// TIA Portal V19 export
FUNCTION "MODE" : Void   // FC3, LAD
{ S7_Optimized_Access := 'TRUE' }
// stored: SetENOAutomatically false
   VAR_TEMP   // added for the SCL form of the ladder/FBD networks
      _w1 : Bool;
   END_VAR
BEGIN

REGION Network 1: MANUAL_MODE_SELECTION
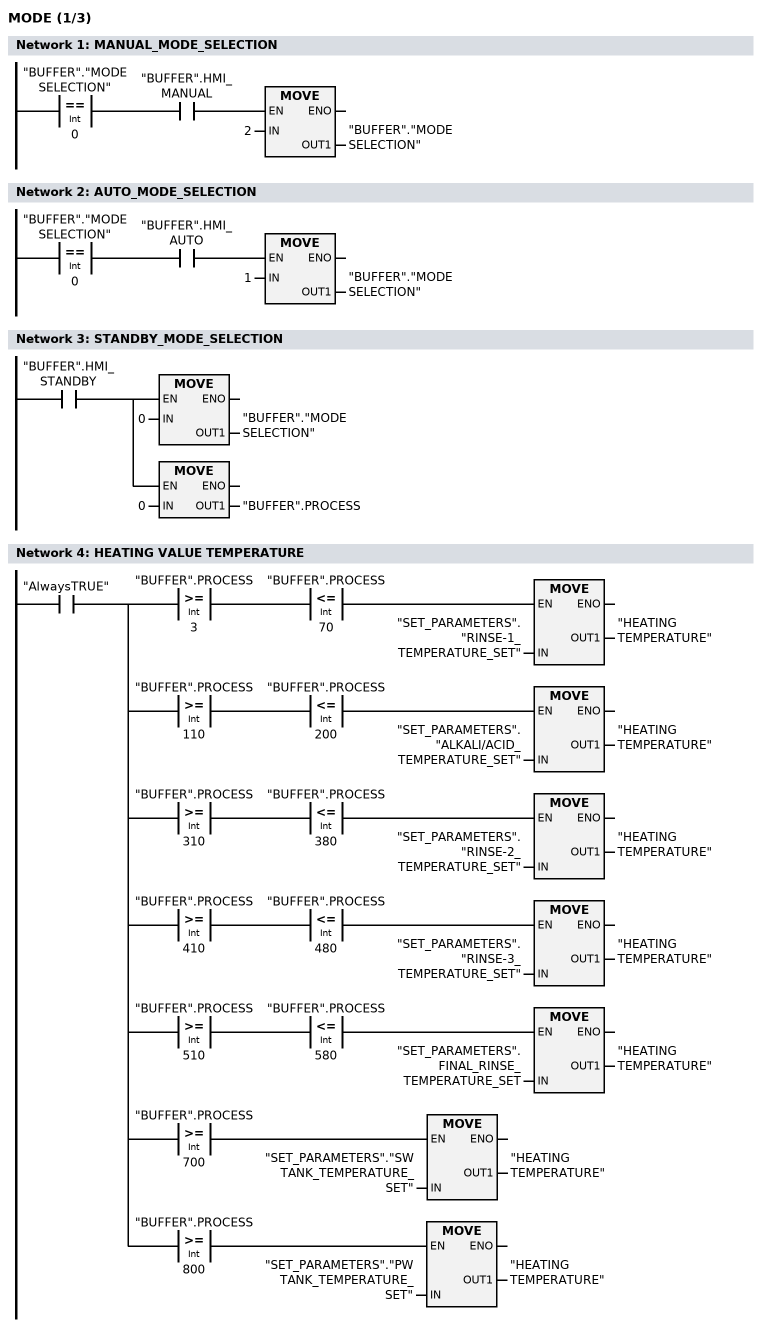
   RUNG wire#powerrail
      { S7_Templates := "SrcType := Int" } EQ_Contact(in1 := "BUFFER"."MODE SELECTION", in2 := 0)
      Contact( "BUFFER".HMI_MANUAL )
      Move(in := 2, out1 => "BUFFER"."MODE SELECTION")
   END_RUNG
   // the same network as SCL:
   IF ("BUFFER"."MODE SELECTION" = 0) AND "BUFFER".HMI_MANUAL THEN "BUFFER"."MODE SELECTION" := 2; END_IF;
END_REGION

REGION Network 2: AUTO_MODE_SELECTION
   RUNG wire#powerrail
      { S7_Templates := "SrcType := Int" } EQ_Contact(in1 := "BUFFER"."MODE SELECTION", in2 := 0)
      Contact( "BUFFER".HMI_AUTO )
      Move(in := 1, out1 => "BUFFER"."MODE SELECTION")
   END_RUNG
   // the same network as SCL:
   IF ("BUFFER"."MODE SELECTION" = 0) AND "BUFFER".HMI_AUTO THEN "BUFFER"."MODE SELECTION" := 1; END_IF;
END_REGION

REGION Network 3: STANDBY_MODE_SELECTION
   RUNG wire#powerrail
      Contact( "BUFFER".HMI_STANDBY )
      wire#w1
      Move(in := 0, out1 => "BUFFER"."MODE SELECTION")
   END_RUNG
   RUNG wire#w1
      Move(in := 0, out1 => "BUFFER".PROCESS)
   END_RUNG
   // the same network as SCL:
   IF "BUFFER".HMI_STANDBY THEN
       "BUFFER"."MODE SELECTION" := 0;
       "BUFFER".PROCESS := 0;
   END_IF;
END_REGION

REGION Network 4: HEATING VALUE TEMPERATURE
   RUNG wire#powerrail
      Contact( "AlwaysTRUE" )
      wire#w1
      { S7_Templates := "SrcType := Int" } GE_Contact(in1 := "BUFFER".PROCESS, in2 := 3)
      { S7_Templates := "SrcType := Int" } LE_Contact(in1 := "BUFFER".PROCESS, in2 := 70)
      Move(in := "SET_PARAMETERS"."RINSE-1_TEMPERATURE_SET", out1 => "HEATING TEMPERATURE")
   END_RUNG
   RUNG wire#w1
      { S7_Templates := "SrcType := Int" } GE_Contact(in1 := "BUFFER".PROCESS, in2 := 110)
      { S7_Templates := "SrcType := Int" } LE_Contact(in1 := "BUFFER".PROCESS, in2 := 200)
      Move(in := "SET_PARAMETERS"."ALKALI/ACID_TEMPERATURE_SET", out1 => "HEATING TEMPERATURE")
   END_RUNG
   RUNG wire#w1
      { S7_Templates := "SrcType := Int" } GE_Contact(in1 := "BUFFER".PROCESS, in2 := 310)
      { S7_Templates := "SrcType := Int" } LE_Contact(in1 := "BUFFER".PROCESS, in2 := 380)
      Move(in := "SET_PARAMETERS"."RINSE-2_TEMPERATURE_SET", out1 => "HEATING TEMPERATURE")
   END_RUNG
   RUNG wire#w1
      { S7_Templates := "SrcType := Int" } GE_Contact(in1 := "BUFFER".PROCESS, in2 := 410)
      { S7_Templates := "SrcType := Int" } LE_Contact(in1 := "BUFFER".PROCESS, in2 := 480)
      Move(in := "SET_PARAMETERS"."RINSE-3_TEMPERATURE_SET", out1 => "HEATING TEMPERATURE")
   END_RUNG
   RUNG wire#w1
      { S7_Templates := "SrcType := Int" } GE_Contact(in1 := "BUFFER".PROCESS, in2 := 510)
      { S7_Templates := "SrcType := Int" } LE_Contact(in1 := "BUFFER".PROCESS, in2 := 580)
      Move(in := "SET_PARAMETERS".FINAL_RINSE_TEMPERATURE_SET, out1 => "HEATING TEMPERATURE")
   END_RUNG
   RUNG wire#w1
      { S7_Templates := "SrcType := Int" } GE_Contact(in1 := "BUFFER".PROCESS, in2 := 700)
      Move(in := "SET_PARAMETERS"."SW TANK_TEMPERATURE_SET", out1 => "HEATING TEMPERATURE")
   END_RUNG
   RUNG wire#w1
      { S7_Templates := "SrcType := Int" } GE_Contact(in1 := "BUFFER".PROCESS, in2 := 800)
      Move(in := "SET_PARAMETERS"."PW TANK_TEMPERATURE_SET", out1 => "HEATING TEMPERATURE")
   END_RUNG
   // the same network as SCL:
   IF "AlwaysTRUE" AND ("BUFFER".PROCESS >= 3) AND ("BUFFER".PROCESS <= 70) THEN
       "HEATING TEMPERATURE" := "SET_PARAMETERS"."RINSE-1_TEMPERATURE_SET";
   END_IF;
   IF "AlwaysTRUE" AND ("BUFFER".PROCESS >= 110) AND ("BUFFER".PROCESS <= 200) THEN
       "HEATING TEMPERATURE" := "SET_PARAMETERS"."ALKALI/ACID_TEMPERATURE_SET";
   END_IF;
   IF "AlwaysTRUE" AND ("BUFFER".PROCESS >= 310) AND ("BUFFER".PROCESS <= 380) THEN
       "HEATING TEMPERATURE" := "SET_PARAMETERS"."RINSE-2_TEMPERATURE_SET";
   END_IF;
   IF "AlwaysTRUE" AND ("BUFFER".PROCESS >= 410) AND ("BUFFER".PROCESS <= 480) THEN
       "HEATING TEMPERATURE" := "SET_PARAMETERS"."RINSE-3_TEMPERATURE_SET";
   END_IF;
   IF "AlwaysTRUE" AND ("BUFFER".PROCESS >= 510) AND ("BUFFER".PROCESS <= 580) THEN
       "HEATING TEMPERATURE" := "SET_PARAMETERS".FINAL_RINSE_TEMPERATURE_SET;
   END_IF;
   IF "AlwaysTRUE" AND ("BUFFER".PROCESS >= 700) THEN
       "HEATING TEMPERATURE" := "SET_PARAMETERS"."SW TANK_TEMPERATURE_SET";
   END_IF;
   IF "AlwaysTRUE" AND ("BUFFER".PROCESS >= 800) THEN
       "HEATING TEMPERATURE" := "SET_PARAMETERS"."PW TANK_TEMPERATURE_SET";
   END_IF;
END_REGION

REGION Network 5: HEATING HYSTERSIS
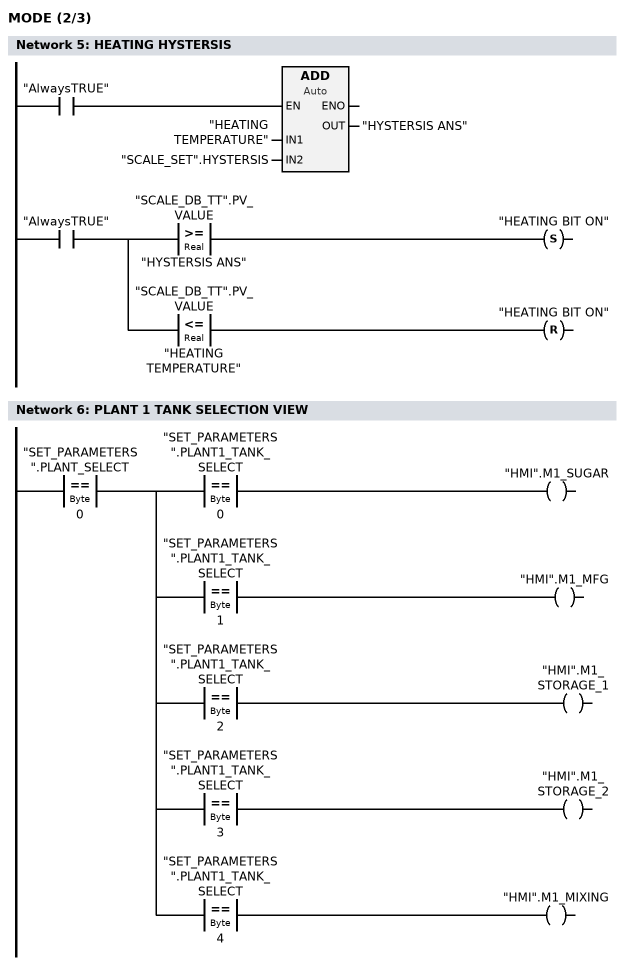
   RUNG wire#powerrail
      Contact( "AlwaysTRUE" )
      Add(in1 := "HEATING TEMPERATURE", in2 := "SCALE_SET".HYSTERSIS, out => "HYSTERSIS ANS")
   END_RUNG
   RUNG wire#powerrail
      Contact( "AlwaysTRUE" )
      wire#w1
      { S7_Templates := "SrcType := Real" } GE_Contact(in1 := "SCALE_DB_TT".PV_VALUE, in2 := "HYSTERSIS ANS")
      S_Coil( "HEATING BIT ON" )
   END_RUNG
   RUNG wire#w1
      { S7_Templates := "SrcType := Real" } LE_Contact(in1 := "SCALE_DB_TT".PV_VALUE, in2 := "HEATING TEMPERATURE")
      R_Coil( "HEATING BIT ON" )
   END_RUNG
   // the same network as SCL:
   IF "AlwaysTRUE" THEN "HYSTERSIS ANS" := "HEATING TEMPERATURE" + "SCALE_SET".HYSTERSIS; END_IF;
   IF "AlwaysTRUE" AND ("SCALE_DB_TT".PV_VALUE >= "HYSTERSIS ANS") THEN "HEATING BIT ON" := TRUE; END_IF;
   IF "AlwaysTRUE" AND ("SCALE_DB_TT".PV_VALUE <= "HEATING TEMPERATURE") THEN
       "HEATING BIT ON" := FALSE;
   END_IF;
END_REGION

REGION Network 6: PLANT 1 TANK SELECTION VIEW
   RUNG wire#powerrail
      { S7_Templates := "SrcType := Byte" } EQ_Contact(in1 := "SET_PARAMETERS".PLANT_SELECT, in2 := 0)
      wire#w1
      { S7_Templates := "SrcType := Byte" } EQ_Contact(in1 := "SET_PARAMETERS".PLANT1_TANK_SELECT, in2 := 0)
      Coil( "HMI".M1_SUGAR )
   END_RUNG
   RUNG wire#w1
      { S7_Templates := "SrcType := Byte" } EQ_Contact(in1 := "SET_PARAMETERS".PLANT1_TANK_SELECT, in2 := 1)
      Coil( "HMI".M1_MFG )
   END_RUNG
   RUNG wire#w1
      { S7_Templates := "SrcType := Byte" } EQ_Contact(in1 := "SET_PARAMETERS".PLANT1_TANK_SELECT, in2 := 2)
      Coil( "HMI".M1_STORAGE_1 )
   END_RUNG
   RUNG wire#w1
      { S7_Templates := "SrcType := Byte" } EQ_Contact(in1 := "SET_PARAMETERS".PLANT1_TANK_SELECT, in2 := 3)
      Coil( "HMI".M1_STORAGE_2 )
   END_RUNG
   RUNG wire#w1
      { S7_Templates := "SrcType := Byte" } EQ_Contact(in1 := "SET_PARAMETERS".PLANT1_TANK_SELECT, in2 := 4)
      Coil( "HMI".M1_MIXING )
   END_RUNG
   // the same network as SCL:
   #_w1 := "SET_PARAMETERS".PLANT_SELECT = 0;
   "HMI".M1_SUGAR := #_w1 AND ("SET_PARAMETERS".PLANT1_TANK_SELECT = 0);
   "HMI".M1_MFG := #_w1 AND ("SET_PARAMETERS".PLANT1_TANK_SELECT = 1);
   "HMI".M1_STORAGE_1 := #_w1 AND ("SET_PARAMETERS".PLANT1_TANK_SELECT = 2);
   "HMI".M1_STORAGE_2 := #_w1 AND ("SET_PARAMETERS".PLANT1_TANK_SELECT = 3);
   "HMI".M1_MIXING := #_w1 AND ("SET_PARAMETERS".PLANT1_TANK_SELECT = 4);
END_REGION

REGION Network 7: PLANT 2 TANK SELECTION VIEW
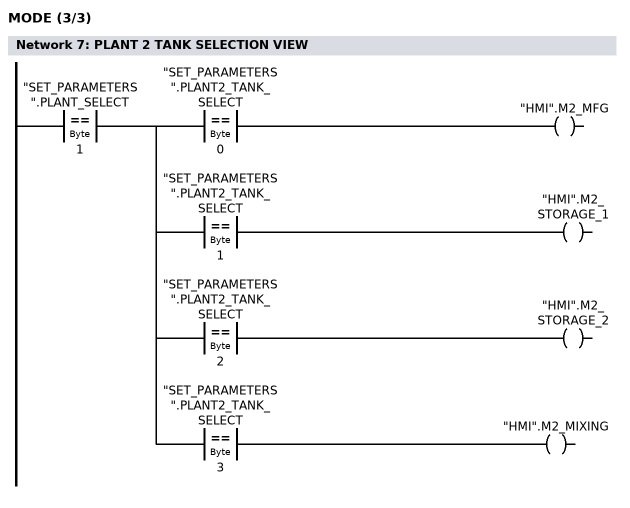
   RUNG wire#powerrail
      { S7_Templates := "SrcType := Byte" } EQ_Contact(in1 := "SET_PARAMETERS".PLANT_SELECT, in2 := 1)
      wire#w1
      { S7_Templates := "SrcType := Byte" } EQ_Contact(in1 := "SET_PARAMETERS".PLANT2_TANK_SELECT, in2 := 0)
      Coil( "HMI".M2_MFG )
   END_RUNG
   RUNG wire#w1
      { S7_Templates := "SrcType := Byte" } EQ_Contact(in1 := "SET_PARAMETERS".PLANT2_TANK_SELECT, in2 := 1)
      Coil( "HMI".M2_STORAGE_1 )
   END_RUNG
   RUNG wire#w1
      { S7_Templates := "SrcType := Byte" } EQ_Contact(in1 := "SET_PARAMETERS".PLANT2_TANK_SELECT, in2 := 2)
      Coil( "HMI".M2_STORAGE_2 )
   END_RUNG
   RUNG wire#w1
      { S7_Templates := "SrcType := Byte" } EQ_Contact(in1 := "SET_PARAMETERS".PLANT2_TANK_SELECT, in2 := 3)
      Coil( "HMI".M2_MIXING )
   END_RUNG
   // the same network as SCL:
   #_w1 := "SET_PARAMETERS".PLANT_SELECT = 1;
   "HMI".M2_MFG := #_w1 AND ("SET_PARAMETERS".PLANT2_TANK_SELECT = 0);
   "HMI".M2_STORAGE_1 := #_w1 AND ("SET_PARAMETERS".PLANT2_TANK_SELECT = 1);
   "HMI".M2_STORAGE_2 := #_w1 AND ("SET_PARAMETERS".PLANT2_TANK_SELECT = 2);
   "HMI".M2_MIXING := #_w1 AND ("SET_PARAMETERS".PLANT2_TANK_SELECT = 3);
END_REGION
END_FUNCTION
